{attribute 'qualified_only'}
{attribute 'strict'}
{attribute 'to_string'}
TYPE e_Jog_Site_Select :
(
	Input_site := 0,
	Output_Site := 1
) INT ;
END_TYPE

(* stored: Version 1.1.0.1, ProductVersion 3.1.4026.13
   EnumerationTextList e_Site_Select: Id {46688c42-71a1-4e19-837b-11f1bdd5e027} *)
